# EPICS substitutions: mpgSupport/Db/ioc/evgPatternIN20.substitutions
file mpgPattern.db
{
#                                  Check    Trigger
#          Device                PNET Data  Seq Ram
  pattern { DEVICE        , SYSI , CHECKI , SENDI }
          { IOC:IN20:EV01 , SYS0 ,   1    ,   0   }
}
file bsaEdefAll.db {
  pattern { DEVICE        , SYSI }
 	  { IOC:IN20:EV01 , SYS0 }
}
file evrPatternAll.db {
#	    Device        , Time Slot Processing         PNET Processing     BSA Data Processing
  pattern { DEVICE        ,         LINK4             ,      LINK5         ,      LINK6           , LINKD }
	  { IOC:IN20:EV01 , IOC:IN20:EV01:TIMESLOTN-1 , IOC:IN20:EV01:PNET , IOC:IN20:EV01:EDEFFO ,  ""   }
}
